// TIA Portal project "HONGPHUONGCAU3TRAM3" (V16)

(* hardware
DEVICE "S7-1200 station_1"  S7-1200 Station
   slot 0: "Rack_0"  S7-1200 Rack  Rack  V1.0
   slot 1: "PLC_1"  CPU 1212C DC/DC/DC  6ES7 212-1AE40-0XB0  V4.3
   slot 2: "DI 16/DQ 16x24VDC_1"  6ES7 223-1BL32-0XB0  V2.0
   slot 3: "DQ 16xRelay_1"  SM 1222 DQ16 x relay  6ES7 222-1HH32-0XB0  V2.0
*)

// ===== PLC "PLC_1"  CPU 1212C DC/DC/DC =====

VAR_GLOBAL   // PLC tag table "Default tag table"
   "Tag_1" AT %I0.0 : Bool;
   "Tag_2" AT %I0.5 : Bool;
   "Tag_3" AT %M0.0 : Bool;
   "KM6" AT %Q0.0 : Bool;
   "KM7(1)" AT %Q1.1 : Bool;
   "KM5" AT %Q0.4 : Bool;
   "KM7" AT %Q0.5 : Bool;
   "Tag_8" AT %M0.3 : Bool;
   "Tag_9" AT %M0.4 : Bool;
END_VAR

// folder: System blocks/Program resources

DATA_BLOCK "T1"   // DB1
{ S7_Optimized_Access := 'TRUE' }
AUTHOR : Simatic
FAMILY : IEC
NAME : IEC_TMR
VERSION : 1.0
// stored: InstanceOfName IEC_TIMER
"IEC_TIMER"
BEGIN
END_DATA_BLOCK

// folder: (top level)

ORGANIZATION_BLOCK "Main"   // OB1, LAD, ProgramCycle
TITLE = "Main Program Sweep (Cycle)"
{ S7_Optimized_Access := 'TRUE' }
VERSION : 0.1
   VAR_INPUT
      Initial_Call : Bool;   // Initial call of this OB
      Remanence : Bool;   // =True, if remanent data are available
   END_VAR
BEGIN

REGION Network 1
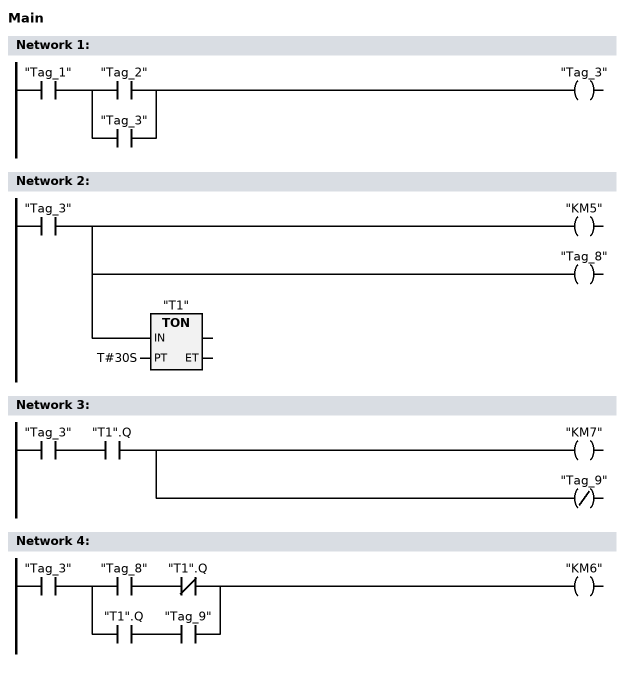
   RUNG wire#powerrail
      Contact( "Tag_1" )
      wire#w1
      Contact( "Tag_2" )
      wire#w2
      Coil( "Tag_3" )
   END_RUNG
   RUNG wire#w1
      Contact( "Tag_3" )
   END_RUNG wire#w2
   // the same network as SCL:
   "Tag_3" := "Tag_1" AND ("Tag_2" OR "Tag_3");
END_REGION

REGION Network 2
   "KM5" := "Tag_3";
   "Tag_8" := "Tag_3";
   "T1".TON(IN := "Tag_3", PT := T#30S);
END_REGION

REGION Network 3
   RUNG wire#powerrail
      Contact( "Tag_3" )
      Contact( "T1".Q )
      wire#w1
      Coil( "KM7" )
   END_RUNG
   RUNG wire#w1
      I_Coil( "Tag_9" )
   END_RUNG
   // the same network as SCL:
   "KM7" := "Tag_3" AND "T1".Q;
   "Tag_9" := NOT "KM7";
END_REGION

REGION Network 4
   RUNG wire#powerrail
      Contact( "Tag_3" )
      wire#w1
      Contact( "Tag_8" )
      I_Contact( "T1".Q )
      wire#w2
      Coil( "KM6" )
   END_RUNG
   RUNG wire#w1
      Contact( "T1".Q )
      Contact( "Tag_9" )
   END_RUNG wire#w2
   // the same network as SCL:
   "KM6" := "Tag_3" AND (("Tag_8" AND NOT "T1".Q) OR ("T1".Q AND "Tag_9"));
END_REGION
END_ORGANIZATION_BLOCK